PROGRAM PRG_IO_Link_Master
VAR
	fbColorSensor			:FB_ColourSensor;
END_VAR

fbColorSensor();

END_PROGRAM

(* stored: Version 1.1.0.1, ProductVersion 3.1.4024.12
   POU PRG_IO_Link_Master: Id {56aa628f-13d5-4975-a6d4-9d393fe72c7e}, SpecialFunc None *)
